(*
    This testsuite tests the different assert-functions for all the primitive data types in TwinCAT, but using the
    ANY-version of the Assert-method.
    For every data type at least two different tests have been defined:
        1. One test that succeeds (Expected and actual are equal)
        2. One test that fails (Expected and actual are false).
    For every failing test the printed value should be the same as if we were using the primitive data type assert
    directly. 
*)
FUNCTION_BLOCK FB_AnyPrimitiveTypes EXTENDS TcUnit.FB_TestSuite

Test_ANY_BYTE_Equals();
Test_ANY_BYTE_Differ();
Test_ANY_BOOL_Equals();
Test_ANY_BOOL_Differ();
Test_ANY_DATE_Equals();
Test_ANY_DATE_Differ();
Test_ANY_DATE_AND_TIME_Equals();
Test_ANY_DATE_AND_TIME_Differ();
Test_ANY_DINT_Equals();
Test_ANY_DINT_Differ();
Test_ANY_DWORD_Equals();
Test_ANY_DWORD_Differ();
Test_ANY_INT_Equals();
Test_ANY_INT_Differ();
Test_ANY_LINT_Equals();
Test_ANY_LINT_Differ();
Test_ANY_LREAL_Equals();
Test_ANY_LREAL_Differ();
Test_ANY_LTIME_Equals();
Test_ANY_LTIME_Differ();
Test_ANY_LWORD_Equals();
Test_ANY_LWORD_Differ();
Test_ANY_REAL_Equals();
Test_ANY_REAL_Differ();
Test_ANY_SINT_Equals();
Test_ANY_SINT_Differ();
Test_ANY_STRING_Equals();
Test_ANY_STRING_Differ();
Test_ANY_STRING_Differ_2();
Test_ANY_TIME_Equals();
Test_ANY_TIME_Differ();
Test_ANY_TIME_OF_DAY_Equals();
TesT_ANY_TIME_OF_DAY_Differ();
Test_ANY_UDINT_Equals();
Test_ANY_UDINT_Differ();
Test_ANY_UINT_Equals();
Test_ANY_UINT_Differ();
Test_ANY_ULINT_Equals();
Test_ANY_ULINT_Differ();
Test_ANY_USINT_Equals();
Test_ANY_USINT_Differ();
Test_ANY_WORD_Equals();
Test_ANY_WORD_Differ();
Test_ANY_WSTRING_Equals();
Test_ANY_WSTRING_Differ();
Test_ANY_WSTRING_Differ_2();

METHOD PRIVATE Test_ANY_BOOL_Differ
VAR
    a : BOOL := TRUE;
    b : BOOL := FALSE;
END_VAR
TEST('Test_ANY_BOOL_Differ');

AssertEquals(Expected := a,
             Actual := b,
             Message := 'Values differ');

TEST_FINISHED();
END_METHOD

METHOD PRIVATE Test_ANY_BOOL_Equals
VAR
    a : BOOL := TRUE;
    b : BOOL := TRUE;
END_VAR
TEST('Test_ANY_BOOL_Equals');

AssertEquals(Expected := a,
             Actual := b,
             Message := 'Values differ');

TEST_FINISHED();
END_METHOD

METHOD PRIVATE Test_ANY_BYTE_Differ
VAR
    a : BYTE := 16#AB;
    b : BYTE := 16#CD;
END_VAR
TEST('Test_ANY_BYTE_Differ');

AssertEquals(Expected := a,
             Actual := b,
             Message := 'Values differ');

TEST_FINISHED();
END_METHOD

METHOD PRIVATE Test_ANY_BYTE_Equals
VAR
    a : BYTE := 16#CD;
    b : BYTE := 16#CD;
END_VAR
TEST('Test_ANY_BYTE_Equals');

AssertEquals(Expected := a,
             Actual := b,
             Message := 'Values differ');

TEST_FINISHED();
END_METHOD

METHOD PRIVATE Test_ANY_DATE_AND_TIME_Differ
VAR
    a : DATE_AND_TIME := DATE_AND_TIME#1996-05-06-15:36:30;
    b : DATE_AND_TIME := DATE_AND_TIME#1972-03-29-00:00:00;
END_VAR
TEST('Test_ANY_DATE_AND_TIME_Differ');

AssertEquals(Expected := a,
             Actual := b,
             Message := 'Values differ');

TEST_FINISHED();
END_METHOD

METHOD PRIVATE Test_ANY_DATE_AND_TIME_Equals
VAR
    a : DATE_AND_TIME := DATE_AND_TIME#2019-01-20-13:54:30;
    b : DATE_AND_TIME := DATE_AND_TIME#2019-01-20-13:54:30;
END_VAR
TEST('Test_ANY_DATE_AND_TIME_Equals');

AssertEquals(Expected := a,
             Actual := b,
             Message := 'Values differ');

TEST_FINISHED();
END_METHOD

METHOD PRIVATE Test_ANY_DATE_Differ
VAR
    a : DATE := DATE#1996-05-06;
    b : DATE := DATE#2019-01-20;
END_VAR
TEST('Test_ANY_DATE_Differ');

AssertEquals(Expected := a,
             Actual := b,
             Message := 'Values differ');

TEST_FINISHED();
END_METHOD

METHOD PRIVATE Test_ANY_DATE_Equals
VAR
    a : DATE := DATE#1996-05-06;
    b : DATE := DATE#1996-05-06;
END_VAR
TEST('Test_ANY_DATE_Equals');

AssertEquals(Expected := a,
             Actual := b,
             Message := 'Values differ');

TEST_FINISHED();
END_METHOD

METHOD PRIVATE Test_ANY_DINT_Differ
VAR
    a : DINT := -55555;
    b : DINT := 70000;
END_VAR
TEST('Test_ANY_DINT_Differ');

AssertEquals(Expected := a,
             Actual := b,
             Message := 'Values differ');

TEST_FINISHED();
END_METHOD

METHOD PRIVATE Test_ANY_DINT_Equals
VAR
    a : DINT := -80000;
    b : DINT := -80000;
END_VAR
TEST('Test_ANY_DINT_Equals');

AssertEquals(Expected := a,
             Actual := b,
             Message := 'Values differ');

TEST_FINISHED();
END_METHOD

METHOD PRIVATE Test_ANY_DWORD_Differ
VAR
    a : DWORD := 16#12345678;
    b : DWORD := 16#90ABCDEF;
END_VAR
TEST('Test_ANY_DWORD_Differ');

AssertEquals(Expected := a,
             Actual := b,
             Message := 'Values differ');

TEST_FINISHED();
END_METHOD

METHOD PRIVATE Test_ANY_DWORD_Equals
VAR
    a : DWORD := 16#7890ABCD;
    b : DWORD := 16#7890ABCD;
END_VAR
TEST('Test_ANY_DWORD_Equals');

AssertEquals(Expected := a,
             Actual := b,
             Message := 'Values differ');

TEST_FINISHED();
END_METHOD

METHOD PRIVATE Test_ANY_INT_Differ
VAR
    a : INT := -32000;
    b : INT := 15423;
END_VAR
TEST('Test_ANY_INT_Differ');

AssertEquals(Expected := a,
             Actual := b,
             Message := 'Values differ');

TEST_FINISHED();
END_METHOD

METHOD PRIVATE Test_ANY_INT_Equals
VAR
    a : INT := -12345;
    b : INT := -12345;
END_VAR
TEST('Test_ANY_INT_Equals');

AssertEquals(Expected := a,
             Actual := b,
             Message := 'Values differ');

TEST_FINISHED();
END_METHOD

METHOD PRIVATE Test_ANY_LINT_Differ
VAR
    a : LINT := -451416345;
    b : LINT := 589532453;
END_VAR
TEST('Test_ANY_LINT_Differ');

AssertEquals(Expected := a,
             Actual := b,
             Message := 'Values differ');

TEST_FINISHED();
END_METHOD

METHOD PRIVATE Test_ANY_LINT_Equals
VAR
    a : LINT := -123456789;
    b : LINT := -123456789;
END_VAR
TEST('Test_ANY_LINT_Equals');

AssertEquals(Expected := a,
             Actual := b,
             Message := 'Values differ');

TEST_FINISHED();
END_METHOD

METHOD PRIVATE Test_ANY_LREAL_Differ
VAR
    a : LREAL := 1234567.89;
    b : LREAL := 1234567.76;
    c : LREAL := 0.0;
END_VAR
TEST('Test_ANY_LREAL_Differ');

AssertEquals(Expected := a,
             Actual := b,
             Message := 'Values a and b differ');

MEMSET (ADR(c), 255, SIZEOF(c));

AssertEquals(Expected := a,
             Actual := c,
             Message := 'Values a and c differ');

TEST_FINISHED();
END_METHOD

METHOD PRIVATE Test_ANY_LREAL_Equals
VAR
    a : LREAL := 1234567.89;
    b : LREAL := 1234567.89;
END_VAR
TEST('Test_ANY_LREAL_Equals');

AssertEquals(Expected := a,
             Actual := b,
             Message := 'Values differ');

TEST_FINISHED();
END_METHOD

METHOD PRIVATE Test_ANY_LTIME_Differ
VAR
    a : LTIME := LTIME#213503D23H34M33S709MS551US615NS;
    b : LTIME := LTIME#1000D15H23M12S34MS2US44NS;
END_VAR
TEST('Test_ANY_LTIME_Differ');

AssertEquals(Expected := a,
             Actual := b,
             Message := 'Values differ');

TEST_FINISHED();
END_METHOD

METHOD PRIVATE Test_ANY_LTIME_Equals
VAR
    a : LTIME := LTIME#213503D23H34M33S709MS551US615NS;
    b : LTIME := LTIME#213503D23H34M33S709MS551US615NS;
END_VAR
TEST('Test_ANY_LTIME_Equals');

AssertEquals(Expected := a,
             Actual := b,
             Message := 'Values differ');

TEST_FINISHED();
END_METHOD

METHOD PRIVATE Test_ANY_LWORD_Differ
VAR
    a : LWORD := 16#0123656789ABCBEC;
    b : LWORD := 16#0123256789ABCAEE;
END_VAR
TEST('Test_ANY_LWORD_Differ');

AssertEquals(Expected := a,
             Actual := b,
             Message := 'Values differ');

TEST_FINISHED();
END_METHOD

METHOD PRIVATE Test_ANY_LWORD_Equals
VAR
    a : LWORD := 16#0123456789ABCDEF;
    b : LWORD := 16#0123456789ABCDEF;
END_VAR
TEST('Test_ANY_LWORD_Equals');

AssertEquals(Expected := a,
             Actual := b,
             Message := 'Values differ');

TEST_FINISHED();
END_METHOD

METHOD PRIVATE Test_ANY_REAL_Differ
VAR
    a : REAL := 1234.5;
    b : REAL := 1234.4;
    c : LREAL := 0.0;
END_VAR
TEST('Test_ANY_REAL_Differ');

AssertEquals(Expected := a,
             Actual := b,
             Message := 'Values a and b differ');

MEMSET (ADR(c), 255, SIZEOF(c));

AssertEquals(Expected := a,
             Actual := c,
             Message := 'Values a and c differ');

TEST_FINISHED();
END_METHOD

METHOD PRIVATE Test_ANY_REAL_Equals
VAR
    a : REAL := 1234.5;
    b : REAL := 1234.5;
END_VAR
TEST('Test_ANY_REAL_Equals');

AssertEquals(Expected := a,
             Actual := b,
             Message := 'Values differ');

TEST_FINISHED();
END_METHOD

METHOD PRIVATE Test_ANY_SINT_Differ
VAR
    a : SINT := 127;
    b : SINT := -30;
END_VAR
TEST('Test_ANY_SINT_Differ');

AssertEquals(Expected := a,
             Actual := b,
             Message := 'Values differ');

TEST_FINISHED();
END_METHOD

METHOD PRIVATE Test_ANY_SINT_Equals
VAR
    a : SINT := -128;
    b : SINT := -128;
END_VAR
TEST('Test_ANY_SINT_Equals');

AssertEquals(Expected := a,
             Actual := b,
             Message := 'Values differ');

TEST_FINISHED();
END_METHOD

METHOD PRIVATE Test_ANY_STRING_Differ
VAR
    a : STRING := 'This is a string';
    b : STRING := 'This is another string';
END_VAR
TEST('Test_ANY_STRING_Differ');

AssertEquals(Expected := a,
             Actual := b,
             Message := 'Values differ');

TEST_FINISHED();
END_METHOD

METHOD PRIVATE Test_ANY_STRING_Differ_2
VAR
    a : STRING := 'This is a string';
    b : STRING := 'This is b string';
END_VAR
TEST('Test_ANY_STRING_Differ_2');

AssertEquals(Expected := a,
             Actual := b,
             Message := 'Values differ');

TEST_FINISHED();
END_METHOD

METHOD PRIVATE Test_ANY_STRING_Equals
VAR
    a : STRING := 'Hello there';
    b : STRING := 'Hello there';
END_VAR
TEST('Test_ANY_STRING_Equals');

AssertEquals(Expected := a,
             Actual := b,
             Message := 'Values differ');

TEST_FINISHED();
END_METHOD

METHOD PRIVATE Test_ANY_TIME_Differ
VAR
    a : TIME := T#12H34M15S10MS;
    b : TIME := T#11H34M13S244MS;
END_VAR
TEST('Test_ANY_TIME_Differ');

AssertEquals(Expected := a,
             Actual := b,
             Message := 'Values differ');

TEST_FINISHED();
END_METHOD

METHOD PRIVATE Test_ANY_TIME_Equals
VAR
    a : TIME := T#11H34M13S244MS;
    b : TIME := T#11H34M13S244MS;
END_VAR
TEST('Test_ANY_TIME_Equals');

AssertEquals(Expected := a,
             Actual := b,
             Message := 'Values differ');

TEST_FINISHED();
END_METHOD

METHOD PRIVATE Test_ANY_TIME_OF_DAY_Differ
VAR
    a : TIME_OF_DAY := TIME_OF_DAY#15:36:30.123;
    b : TIME_OF_DAY := TIME_OF_DAY#06:21:11.492;
END_VAR
TEST('Test_ANY_TIME_OF_DAY_Differ');

AssertEquals(Expected := a,
             Actual := b,
             Message := 'Values differ');

TEST_FINISHED();
END_METHOD

METHOD PRIVATE Test_ANY_TIME_OF_DAY_Equals
VAR
    a : TIME_OF_DAY := TIME_OF_DAY#06:21:11.492;
    b : TIME_OF_DAY := TIME_OF_DAY#06:21:11.492;
END_VAR
TEST('Test_ANY_TIME_OF_DAY_Equals');

AssertEquals(Expected := a,
             Actual := b,
             Message := 'Values differ');

TEST_FINISHED();
END_METHOD

METHOD PRIVATE Test_ANY_UDINT_Differ
VAR
    a : UDINT := 34124214;
    b : UDINT := 52343244;
END_VAR
TEST('Test_ANY_UDINT_Differ');

AssertEquals(Expected := a,
             Actual := b,
             Message := 'Values differ');

TEST_FINISHED();
END_METHOD

METHOD PRIVATE Test_ANY_UDINT_Equals
VAR
    a : UDINT := 21845123;
    b : UDINT := 21845123;
END_VAR
TEST('Test_ANY_UDINT_Equals');

AssertEquals(Expected := a,
             Actual := b,
             Message := 'Values differ');

TEST_FINISHED();
END_METHOD

METHOD PRIVATE Test_ANY_UINT_Differ
VAR
    a : UINT := 64322;
    b : UINT := 32312;
END_VAR
TEST('Test_ANY_UINT_Differ');

AssertEquals(Expected := a,
             Actual := b,
             Message := 'Values differ');

TEST_FINISHED();
END_METHOD

METHOD PRIVATE Test_ANY_UINT_Equals
VAR
    a : UINT := 65535;
    b : UINT := 65535;
END_VAR
TEST('Test_ANY_UINT_Equals');

AssertEquals(Expected := a,
             Actual := b,
             Message := 'Values differ');

TEST_FINISHED();
END_METHOD

METHOD PRIVATE Test_ANY_ULINT_Differ
VAR
    a : ULINT := 10000;
    b : ULINT := 53685437234;
END_VAR
TEST('Test_ANY_ULINT_Differ');

AssertEquals(Expected := a,
             Actual := b,
             Message := 'Values differ');

TEST_FINISHED();
END_METHOD

METHOD PRIVATE Test_ANY_ULINT_Equals
VAR
    a : ULINT := 45683838383;
    b : ULINT := 45683838383;
END_VAR
TEST('Test_ANY_ULINT_Equals');

AssertEquals(Expected := a,
             Actual := b,
             Message := 'Values differ');

TEST_FINISHED();
END_METHOD

METHOD PRIVATE Test_ANY_USINT_Differ
VAR
    a : USINT := 3;
    b : USINT := 7;
END_VAR
TEST('Test_ANY_USINT_Differ');

AssertEquals(Expected := a,
             Actual := b,
             Message := 'Values differ');

TEST_FINISHED();
END_METHOD

METHOD PRIVATE Test_ANY_USINT_Equals
VAR
    a : USINT := 5;
    b : USINT := 5;
END_VAR
TEST('Test_ANY_USINT_Equals');

AssertEquals(Expected := a,
             Actual := b,
             Message := 'Values differ');

TEST_FINISHED();
END_METHOD

METHOD PRIVATE Test_ANY_WORD_Differ
VAR
    a : WORD := 16#EF01;
    b : WORD := 16#2345;
END_VAR
TEST('Test_ANY_WORD_Differ');

AssertEquals(Expected := a,
             Actual := b,
             Message := 'Values differ');

TEST_FINISHED();
END_METHOD

METHOD PRIVATE Test_ANY_WORD_Equals
VAR
    a : WORD := 16#ABCD;
    b : WORD := 16#ABCD;
END_VAR
TEST('Test_ANY_WORD_Equals');

AssertEquals(Expected := a,
             Actual := b,
             Message := 'Values differ');

TEST_FINISHED();
END_METHOD

METHOD PRIVATE Test_ANY_WSTRING_Differ
VAR
    a : WSTRING := "äö";
    b : WSTRING := "æå";
END_VAR
TEST('Test_ANY_WSTRING_Differ');

AssertEquals(Expected := a,
             Actual := b,
             Message := 'Values differ');

TEST_FINISHED();
END_METHOD

METHOD PRIVATE Test_ANY_WSTRING_Differ_2
VAR
    a : WSTRING := "äö◦";
    b : WSTRING := "æå";
END_VAR
TEST('Test_ANY_WSTRING_Differ_2');

AssertEquals(Expected := a,
             Actual := b,
             Message := 'Values differ');

TEST_FINISHED();
END_METHOD

METHOD PRIVATE Test_ANY_WSTRING_Equals
VAR
    a : WSTRING := "ĠĦ";
    b : WSTRING := "ĠĦ";
END_VAR
TEST('Test_ANY_WSTRING_Equals');

AssertEquals(Expected := a,
             Actual := b,
             Message := 'Values differ');

TEST_FINISHED();
END_METHOD

END_FUNCTION_BLOCK

(* stored: Version 1.1.0.1
   POU FB_AnyPrimitiveTypes: Id {bf0ad75f-805b-4448-a5e9-9fafb9350eaa}, SpecialFunc None
   Method Test_ANY_BOOL_Differ: Id {9def4202-9b1d-4fca-a694-7baecaa73c6d}
   Method Test_ANY_BOOL_Equals: Id {24b88842-0df5-436f-8f65-86f62612214c}
   Method Test_ANY_BYTE_Differ: Id {dd37329d-bb06-4679-abf4-e4d04399c232}
   Method Test_ANY_BYTE_Equals: Id {2f42883b-2905-4fcf-ab87-5d19e1fac7b2}
   Method Test_ANY_DATE_AND_TIME_Differ: Id {0d3f804a-d51e-43e6-bd81-f031ee7308e1}
   Method Test_ANY_DATE_AND_TIME_Equals: Id {3b6f68a1-4ae4-42ef-9963-3b1290dfe7f6}
   Method Test_ANY_DATE_Differ: Id {cfc83bfe-e5f8-4bb0-9243-3c64bb120dae}
   Method Test_ANY_DATE_Equals: Id {d466f1ae-1c99-4517-81d7-ba44ee80c32f}
   Method Test_ANY_DINT_Differ: Id {cb70e186-1a96-4b29-985d-60f5f4684775}
   Method Test_ANY_DINT_Equals: Id {ac4e8032-dccc-4a7e-9803-44020c8533e4}
   Method Test_ANY_DWORD_Differ: Id {23ed3054-fb0f-4676-a33d-13cb685f2f27}
   Method Test_ANY_DWORD_Equals: Id {5708854e-5f0b-4ac2-80a1-0b3d9009a3ed}
   Method Test_ANY_INT_Differ: Id {3902bfc9-94f5-457a-8cf1-bf8e15c96e38}
   Method Test_ANY_INT_Equals: Id {16ed816c-bec6-46ce-a406-42d965e0fb31}
   Method Test_ANY_LINT_Differ: Id {fb115c0d-34a2-4d3c-af00-30e036afd5d7}
   Method Test_ANY_LINT_Equals: Id {668fbd05-1b2c-4b08-8d52-d1aaaa059802}
   Method Test_ANY_LREAL_Differ: Id {c7618ef1-aae1-478a-8d43-1bb5a958b641}
   Method Test_ANY_LREAL_Equals: Id {d886c391-4ffc-42ba-aacc-8f8f2b3a5e54}
   Method Test_ANY_LTIME_Differ: Id {c72b07c9-bd17-4b41-8647-93f2630ffe0c}
   Method Test_ANY_LTIME_Equals: Id {ccdb0dec-fafe-402a-802f-577154e15f12}
   Method Test_ANY_LWORD_Differ: Id {ef3f03f1-1a53-4489-8c36-c28660c1e7b7}
   Method Test_ANY_LWORD_Equals: Id {19993f03-49d7-4cee-97a1-88ff9d9eb2e6}
   Method Test_ANY_REAL_Differ: Id {f2472e3d-089e-474c-b4b8-54a3d353ad64}
   Method Test_ANY_REAL_Equals: Id {8290f811-4b5b-4e83-b6ee-422a2bd05e2b}
   Method Test_ANY_SINT_Differ: Id {b0f8ac71-681f-4f1a-94dd-32b085f23744}
   Method Test_ANY_SINT_Equals: Id {630cc9a7-6d4d-40eb-ab44-a0a4844068f6}
   Method Test_ANY_STRING_Differ: Id {8384ce7c-1f54-4249-9dc0-3b2f1dfa1e90}
   Method Test_ANY_STRING_Differ_2: Id {1979c19d-5f81-4ca1-b2ab-1e735e3c2f9f}
   Method Test_ANY_STRING_Equals: Id {45fb731e-62a5-4739-983d-66e18d9850be}
   Method Test_ANY_TIME_Differ: Id {361fa935-4959-4eb6-b25a-f9965f1f30dd}
   Method Test_ANY_TIME_Equals: Id {8b715def-1875-46d4-8b4b-cd8cbb83966f}
   Method Test_ANY_TIME_OF_DAY_Differ: Id {6a1b7492-d6c5-4590-b52d-c2c8e1ee1844}
   Method Test_ANY_TIME_OF_DAY_Equals: Id {54c634d0-a0c1-46c0-81a9-2d082c52fde4}
   Method Test_ANY_UDINT_Differ: Id {e30459bf-ebf3-48ab-a1c1-3d0dd57a829e}
   Method Test_ANY_UDINT_Equals: Id {9c466d83-1d0b-48d6-a187-0404dcd7fc0c}
   Method Test_ANY_UINT_Differ: Id {6fcb372c-bdc6-4fa3-bdd8-941d914d6b3a}
   Method Test_ANY_UINT_Equals: Id {9e678934-ef5b-42e1-a53f-17737ee06d35}
   Method Test_ANY_ULINT_Differ: Id {dae19af6-fcc2-42c1-aaca-8dc7c861bdcc}
   Method Test_ANY_ULINT_Equals: Id {f13de1a5-523a-4c9d-8e7e-8c0b2840de93}
   Method Test_ANY_USINT_Differ: Id {feb2c66c-f754-4a55-ba64-e1fdc77ddce6}
   Method Test_ANY_USINT_Equals: Id {44a01ea7-d3cf-4d20-aeb7-e4787721e931}
   Method Test_ANY_WORD_Differ: Id {684677fe-b88b-4336-9954-f4e16d3d3cf5}
   Method Test_ANY_WORD_Equals: Id {962442d1-3576-440d-880d-7ca8abee0ca2}
   Method Test_ANY_WSTRING_Differ: Id {47cc195f-2b65-4c94-84a6-ca1ea74f987f}
   Method Test_ANY_WSTRING_Differ_2: Id {edbbe9e9-fe3b-4d3b-8d0a-cb170d68100f}
   Method Test_ANY_WSTRING_Equals: Id {2359fafa-0714-42b0-8ab4-3be6341813c5} *)
